Staubli VAL3: setList.pgx

public program setList(string x_sTitle (dimensions=1), string& x_sListItem[] (dimensions=1), bool x_bUserRefresh (dimensions=1), bool x_bListItemRef (dimensions=1), num& x_nSelected (dimensions=1), string& x_sItem (dimensions=1), num& x_nKey (dimensions=1))
  local num l_nView
  local num l_nItem
begin
  if x_bUserRefresh
    if x_bListItemRef
      call setSizeList(20,0,18,11)
      call listcreate(x_sTitle)
      if x_sListItem[0]!=""
        call listadd(x_sListItem)
      endIf
    else
      call setSizeList(20,0,18,11)
      call listframe(x_sTitle,nTopX,nTopY,nBottomX,nBottomY)
    endIf
    call selectNewField(x_nSelected,l_nItem,l_nView)
  endIf
  x_nKey=getKey()
  call listevent(x_nKey,l_nItem,x_sItem)
  l_nView=nView
  x_nSelected=l_nItem
end
